// TIA Portal V18 export
// export: Created 2025-12-01T17:51:16.8602364Z, ExportSetting None, DisplayName Totally Integrated Automation Portal, DisplayVersion V18 Update 5, DisplayName TIA Portal Openness, DisplayVersion V18 Update 5, DisplayName TIA Portal Teamcenter Gateway, DisplayVersion V18, DisplayName TIA Portal Version Control Interface, DisplayVersion V18, DisplayName STEP 7 Professional, DisplayVersion V18 Update 5, DisplayName STEP 7 Safety, DisplayVersion V18, DisplayName WinCC Professional, DisplayVersion V18 Update 5
DATA_BLOCK "KeyenceSR1000Ctrl_807A1DB"   // DB1808
// stored: AutoNumber false, InstanceOfName KeyenceSR1000Ctrl, InstanceOfType FB
"KeyenceSR1000Ctrl"
   // VAR_INPUT
   //    iI_Address { ExternalAccessible := 'False'; ExternalVisible := 'False'; ExternalWritable := 'False'} : Int;
   //    iO_Address : Int;
   //    iSysRun : Bool;
   //    iReset : Bool;
   //    iAuto : Bool;
   //    iManual : Bool;
   //    iReTriggerLimitTimes : USInt;
   // END_VAR
   // VAR_OUTPUT
   //    oReady : Bool;
   //    oComplete : Bool;
   //    oError : Bool;
   //    oErrorCode : UInt;
   // END_VAR
   // VAR_IN_OUT
   //    ioAutoTrigger : Bool;
   // END_VAR
   // VAR
   //    sHMI { S7_SetPoint := 'True'} : "RCS_KeyenceSR1000_HMI1";
   //    sCtrl : Struct
   //       Sequence : Int;
   //    END_STRUCT;
   //    sCurrentCode : String[128];
   //    sInData { S7_SetPoint := 'True'} : "RCS_KeyenceSR1000_Input1";
   //    sOutData { S7_SetPoint := 'True'} : "RCS_KeyenceSR1000_Output1";
   //    sAutoOld : Bool;
   //    sManualOld : Bool;
   //    sBusyTimeOut : Bool;
   //    sRunTimer { S7_SetPoint := 'True'} : TON_TIME;
   //    sBusyTimer { S7_SetPoint := 'True'} : TON_TIME;
   //    sFindCurrentPos { S7_SetPoint := 'True'} : Int;
   // END_VAR
BEGIN
END_DATA_BLOCK
